// TIA Portal project "Temporizzatore" (V16)

(* hardware
DEVICE "S7-1200 station_1"  S7-1200 Station
   slot 0: "Telaio di montaggio_0"  S7-1200 Rack  Rack  V1.0
   slot 1: "PLC_1"  CPU 1215C DC/DC/Rly  6ES7 215-1HG40-0XB0  V4.4
*)

// ===== PLC "PLC_1"  CPU 1215C DC/DC/Rly =====

VAR_GLOBAL   // PLC tag table "Tabella delle variabili standard"
   "marcia" AT %I1.0 : Bool;   // attivo quando premuto
   "emergenza" AT %I0.7 : Bool;   // attivo quando non premuto
   "start" AT %I1.1 : Bool;   // attivo quando premuto
   "arresto" AT %I1.2 : Bool;   // attivo quando premuto
   "macchina_on" AT %M0.0 : Bool;   // macchina accesa
   "avanti" AT %Q0.0 : Bool;
   "indietro" AT %Q0.1 : Bool;
   "spia_macchina_on" AT %Q0.6 : Bool;
   "fotocellula1_nastroSemplice" AT %I0.0 : Bool;   // attiva quando non oscurata
   "fotocellula2_nastroSemplice" AT %I0.1 : Bool;   // attiva quando non oscurata
   "contaimpulsi_nastroSemplice" AT %I0.2 : Bool;   // 4 impulsi per giro dell’albero motore
   "fotocellula_3_pressa" AT %I0.3 : Bool;   // oscurata (non attiva) quando si mette un pezzo
   "fotocellula_4_pressa" AT %I0.4 : Bool;   // oscurata (non attiva) quando il pezzo è sotto la
   "fine_corsa_pressa_alta" AT %I0.5 : Bool;   // attivo quando la pressa è in posizione home
   "fine_corsa_pressa_bassa" AT %I0.6 : Bool;   // attivo quando la pressa è tutta giù
   "option" AT %I1.3 : Bool;   // attivo quando premuto
   "S1_selettore_1" AT %I1.4 : Bool;   // attivo in posizione 1
   "S2 selettore 2" AT %I1.5 : Bool;   // attivo in posizione 2
   "SpiaMotoreF1-F2" AT %Q0.7 : Bool;
   "SpiaMotoreF2-F1" AT %Q1.0 : Bool;
END_VAR

// folder: System blocks/Program resources

DATA_BLOCK "Cont_UP"   // DB1
{ S7_Optimized_Access := 'TRUE' }
AUTHOR : Simatic
FAMILY : IEC
NAME : CNTR
VERSION : 1.0
// stored: InstanceOfName IEC_COUNTER
"IEC_COUNTER"
BEGIN
END_DATA_BLOCK

DATA_BLOCK "ContaTempo"   // DB2
{ S7_Optimized_Access := 'TRUE' }
AUTHOR : Simatic
FAMILY : IEC
NAME : IEC_TMR
VERSION : 1.0
// stored: InstanceOfName IEC_TIMER
"IEC_TIMER"
BEGIN
END_DATA_BLOCK

// folder: (top level)

ORGANIZATION_BLOCK "Main"   // OB1, LAD, ProgramCycle
TITLE = "Main Program Sweep (Cycle)"
{ S7_Optimized_Access := 'TRUE' }
VERSION : 0.1
   VAR_INPUT
      Initial_Call : Bool;   // Initial call of this OB
      Remanence : Bool;   // =True, if remanent data are available
   END_VAR
BEGIN

REGION Network 1: Temporizzatore
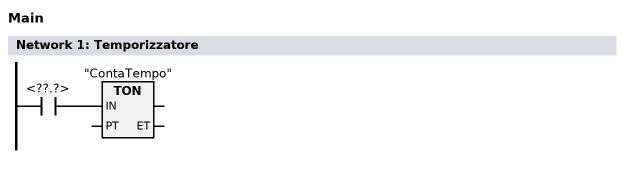
   // no checked SCL form for this network; see the picture
END_REGION
END_ORGANIZATION_BLOCK